PROGRAM MAIN
VAR
	output1 :BOOL;
	input1: BOOL;
	counter : INT;
END_VAR

counter := counter +1;

END_PROGRAM

(* stored: Version 1.1.0.1, ProductVersion 3.1.4024.12
   POU MAIN: Id {3623e513-07cc-4d13-b30e-006b26bc4cde}, SpecialFunc None *)
